PROGRAM main
  VAR
    START AT %IX0.0 : BOOL; (* Start pushbutton, GPIO 18, pull-down. 1 = pressed. *)
    STOP AT %IX0.1 : BOOL; (* Stop pushbutton, GPIO 19, pull-down. 1 = pressed. Used as an NC contact in Rung 1, so pressing it breaks the seal. *)
    LED AT %QX0.0 : BOOL; (* Run indicator LED, GPIO 5. 1 = lit. Flashes while the machine is running. *)
    RUN : BOOL; (* Internal run bit, no physical I/O. 1 = machine running. Set by Start, cleared by Stop (Rung 1). *)
    T1_DONE : BOOL; (* Internal bit. 1 = flasher timer T1 done, LED on phase (Rung 2). *)
    T2_DONE : BOOL; (* Internal bit. 1 = flasher timer T2 done, resets T1 (Rung 3). *)
    T1 : TON; (* Flasher timer 1, TON 500 ms. Times the LED off phase. *)
    T2 : TON; (* Flasher timer 2, TON 500 ms. Times the LED on phase. *)
  END_VAR

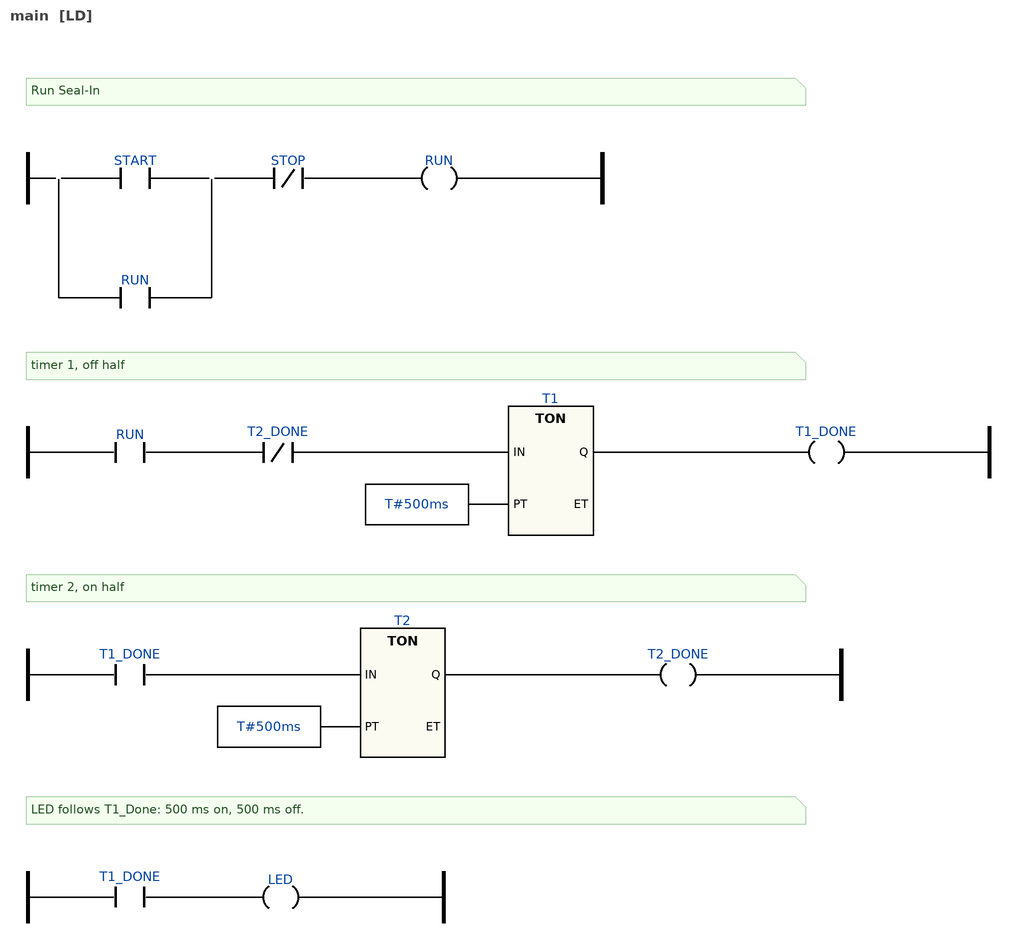
(* LD diagram, written out as Structured Text *)
(* Run Seal-In *)
RUN := (START OR RUN) AND NOT STOP;
(* timer 1, off half *)
T1(IN := RUN AND NOT T2_DONE, PT := T#500ms);
T1_DONE := T1.Q;
(* timer 2, on half *)
T2(IN := T1_DONE, PT := T#500ms);
T2_DONE := T2.Q;
(* LED follows T1_Done: 500 ms on, 500 ms off. *)
LED := T1_DONE;
END_PROGRAM
